(* PLC project TwinForge OpenPLC Smoke Test, TwinForge TwinForge 0.1.0 *)
(* stored: creationDateTime 2026-07-30T00:00:00+00:00 *)

PROGRAM PLC_PRG
  VAR
    Enable : BOOL;
    Output : BOOL;
  END_VAR

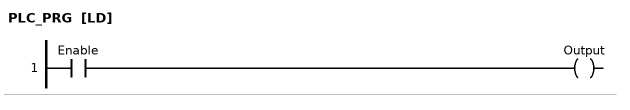
(* LD diagram, written out as Structured Text *)
Output := Enable;
END_PROGRAM

CONFIGURATION OpenPLCSmoke
  RESOURCE Application ON PLC
    TASK MainTask(INTERVAL := T#20ms, PRIORITY := 1);
    PROGRAM PLC_PRG WITH MainTask : PLC_PRG;
  END_RESOURCE
END_CONFIGURATION
